// TwinCAT 3 PLC project B2SignedDelta_Plc
// Title: B2SignedDelta_Plc
// Company: Tc3 Project
// ProjectVersion: 1.0.0.0
// ProgramVersion: 3.1.4026.22
// libraries:
//   Tc2_Standard, * (Beckhoff Automation GmbH)
//   Tc2_System, * (Beckhoff Automation GmbH)
// project tree:
//   / PlcTask.TcTTO
//   POUs/ FB_Counter.TcPOU, MAIN.TcPOU
// real-time tasks:
//   TASK PlcTask: cycle T#10ms, priority 20, ADS port 350

CONFIGURATION B2SignedDelta_Plc
    RESOURCE PLC ON TwinCAT3
        TASK PlcTask(INTERVAL := T#10ms, PRIORITY := 20);
        PROGRAM MAIN WITH PlcTask : MAIN;
    END_RESOURCE
END_CONFIGURATION

// ---- POUs/MAIN.TcPOU
PROGRAM MAIN
VAR
END_VAR

END_PROGRAM

// ---- POUs/FB_Counter.TcPOU
FUNCTION_BLOCK FB_Counter
VAR
END_VAR

METHOD GetSignedDelta : UDINT
VAR_INPUT
    a : INT;
    b : INT;
END_VAR
GetSignedDelta := DINT_TO_UDINT(INT_TO_DINT(a) - INT_TO_DINT(b));
END_METHOD

END_FUNCTION_BLOCK
